Fanuc KAREL source: VT_GET_QUEUE.kl

PROGRAM T
%NOLOCKGROUP
VAR
 v0 : INTEGER
 v1 : INTEGER
 v2 : INTEGER
 v3 : INTEGER
 v4 : INTEGER
 v5 : INTEGER
 v6 : INTEGER
BEGIN
 VT_GET_QUEUE(v0, v1, v2, v3, v4, v5, v6)
END T
